TYPE DiffNumbers :
UNION
	fA : REAL;
    nB : UDINT;
    nC : WORD;
	
END_UNION
END_TYPE

(* stored: Version 1.1.0.1, ProductVersion 3.1.4024.16
   DUT DiffNumbers: Id {5332fbb7-db96-42e4-8e2f-5bce61e53feb} *)
